# EPICS substitutions: pimegaApp/Db/pimega450d.substitutions
file "module.template" {
   pattern { MODULE, ADDR }
           { M1:,    0    }
           { M2:,    1    }
           { M3:,    2    }
           { M4:,    3    }
           { M5:,    4    }
           { M6:,    5    }
           { M7:,    6    }
           { M8:,    7    }
           { M9:,    8    }
           { M10:,   9    }
}
